Staubli VAL3: bin2dec.pgx

public program bin2dec(num& x_nInput[], num& x_nResult)
  local num l_nElement
begin
  x_nResult = 0

  for l_nElement = 0 to size(x_nInput)-1
    x_nResult = x_nResult + x_nInput[l_nElement]*power(2,size(x_nInput) -1-l_nElement)
  endFor

end
